FUNCTION_BLOCK EL2798
VAR
	{attribute addProperty Name "WcState"}
	_wcState : WcStateBase;
	{attribute addProperty Name "Info data"}
	_infoData : InfoDataBase;
	_io : EL2xx8_Data;
END_VAR

PROPERTY IO : REFERENCE TO EL2xx8_Data
GET
IO REF= _io;
END_GET
END_PROPERTY

PROPERTY WcState : REFERENCE TO WcStateBase
GET
WcState REF= _wcState;
END_GET
END_PROPERTY

END_FUNCTION_BLOCK

(* stored: Version 1.1.0.1, ProductVersion 3.1.4024.9
   POU EL2798: Id {187ad276-283f-045e-34a7-2b3d4134ff2c}, SpecialFunc None
   Property IO: Id {807f8380-8053-08f5-1082-59378419008b}
   Get Get: Id {f0f483a5-5162-0a7e-0be9-9fe167a46427}
   Property WcState: Id {ca9adb32-287d-0b15-1d57-20c3c8cc4267}
   Get Get: Id {6ad03371-dd6c-0029-3fc1-24e47be690b5} *)
